FUNCTION_BLOCK TcoSequencerAutoRestorableTest EXTENDS TcoCore._internals_TcoContext
VAR
	_callMyPlcInstance	:	BOOL := FALSE;
	_sequencer : _TcoSequencer(THIS^, NO.Structure, eRestoreMode.AutoRestoreMembers);
	_runPLCinstanceOnce : BOOL := FALSE;
	_runPLCinstanceCyclicaly : BOOL := FALSE;
	_stepID : INT := 32764;
	_enabled : BOOL;
	_stepDescription : STRING := 'Last step sequence message';	
	_runOneStep : BOOL;
	_runAllSteps : BOOL;
	_finishStep : BOOL;
	_restore : BOOL;
	_cycleCount : INT;
	_restoreCycleCount : INT;
	_init: BOOL;
	_setCurrentStepPropTestData : TcoCore.StepDetails;
END_VAR

IF _callMyPlcInstance THEN
	IF NOT _init THEN
		ContextOpen();	
		ContextClose();	
		_init := THIS^._rtc.IsValid;
	END_IF
	
	IF _restore THEN
		ContextOpen();	
		THIS^._sequencer.Restore();	
		_restoreCycleCount := _restoreCycleCount + 1;
		_restore := FALSE;
		ContextClose();	
		RETURN;
	END_IF
	
	IF _runPLCinstanceOnce AND NOT _runPLCinstanceCyclicaly THEN
		ContextOpen();	
		THIS^.PLCinstanceRun(_stepID , _enabled, _stepDescription);
		_cycleCount := _cycleCount + 1;
		_runPLCinstanceOnce := FALSE;
		ContextClose();	
	END_IF
	
	IF _runPLCinstanceCyclicaly AND NOT _runPLCinstanceOnce THEN
		ContextOpen();	
		THIS^.PLCinstanceRun(_stepID , _enabled, _stepDescription);
		_cycleCount := _cycleCount + 1;
		ContextClose();	
	END_IF
END_IF;

{attribute 'TcRpcEnable'}
METHOD ChildHasAutoRestoreEnabled : BOOL;
ChildHasAutoRestoreEnabled := _sequencer.ChildHasAutoRestoreEnabled();
END_METHOD

{attribute 'TcRpcEnable'}
METHOD ChildIsAutoRestorable : BOOL;
ChildIsAutoRestorable := _sequencer.ChildIsAutoRestorable();
END_METHOD

{attribute 'TcRpcEnable'}
METHOD CleanupPointers
_sequencer.CleanupPointers();
END_METHOD

{attribute 'TcRpcEnable'}
METHOD ClearNumberOfSteps
_sequencer.ClearNumberOfSteps();
END_METHOD

{attribute 'TcRpcEnable'}
METHOD PROTECTED ContextClose
SUPER^._Close();
END_METHOD

{attribute 'TcRpcEnable'}
METHOD ContextOpen
SUPER^._Open();
END_METHOD

{attribute 'TcRpcEnable'}
METHOD GetChildState : INT
GetChildState := _sequencer.GetChildState();
END_METHOD

{attribute 'TcRpcEnable'}
METHOD GetCurrentStepOrder : UINT
GetCurrentStepOrder := _sequencer._currentStep.Order;
END_METHOD

{attribute 'TcRpcEnable'}
METHOD GetCurrentStepPropTest
_setCurrentStepPropTestData := THIS^._sequencer.CurrentStep;
END_METHOD

{attribute 'TcRpcEnable'}
METHOD GetNumberOfStepsInSequence : UINT
GetNumberOfStepsInSequence := _sequencer._numberOfStepsInSequence;
END_METHOD

{attribute 'TcRpcEnable'}
METHOD GetOrderOfTheCurrentlyEvaluatedStep : UINT
GetOrderOfTheCurrentlyEvaluatedStep := _sequencer._theOrderOfTheCurrentlyEvaluatedStep;
END_METHOD

{attribute 'TcRpcEnable'}
METHOD GetOrderOfTheCurrentlyExecutedStep : UINT
GetOrderOfTheCurrentlyExecutedStep := _sequencer._theOrderOfTheCurrentlyExecutedStep;
END_METHOD

{attribute 'TcRpcEnable'}
METHOD GetPreviousNumberOfStepsInSequence : UINT
GetPreviousNumberOfStepsInSequence := _sequencer._previousNumberOfStepsInSequence;
END_METHOD

{attribute 'TcRpcEnable'}
METHOD GetRequestStepCycle : UINT
GetRequestStepCycle := _sequencer.RequestStepCycle;
END_METHOD

{attribute 'TcRpcEnable'}
METHOD GetSequencerErrorId : INT
GetSequencerErrorId := _sequencer.GetSequencerErrorId();
END_METHOD

{attribute 'TcRpcEnable'}
METHOD GetTextOfTheMostImportantMessage : STRING(254)
GetTextOfTheMostImportantMessage := THIS^._sequencer.GetTextOfTheMostImportantMessage();
END_METHOD

{attribute 'TcRpcEnable'}
METHOD HasAutoRestoreEnabled : BOOL;
HasAutoRestoreEnabled := _sequencer.HasAutoRestoreEnabled();
END_METHOD

{attribute 'TcRpcEnable'}
METHOD IsAutoRestorable : BOOL;
IsAutoRestorable := _sequencer.IsAutoRestorable();
END_METHOD

{attribute 'TcRpcEnable'}
METHOD IsFirstStepEntry : BOOL
IsFirstStepEntry := THIS^._sequencer.IsFirstStepEntry();
END_METHOD

METHOD PROTECTED  Main
END_METHOD

{attribute 'TcRpcEnable'}
METHOD PLCinstanceRun
VAR_INPUT
	inStepId			:	UINT;
	inEnabled			:	BOOL;
	inStepDescription	:	STRING(254);	
END_VAR
THIS^._sequencer.SetTestParams(	_runOneStep , _runAllSteps , _finishStep , inStepId , inEnabled , inStepDescription);

THIS^._sequencer.Run();
END_METHOD

{attribute 'TcRpcEnable'}
METHOD RequestStep
VAR_INPUT
	inRequestedStepId : INT;
END_VAR
_sequencer._RequestStep(inRequestedStepId);
END_METHOD

{attribute 'TcRpcEnable'}
METHOD Restore
_sequencer.Restore();
END_METHOD

{attribute 'TcRpcEnable'}
METHOD SequenceComplete
_sequencer._SequenceComplete();
END_METHOD

{attribute 'TcRpcEnable'}
METHOD SequencerClose
THIS^._sequencer.SequencerClose();
END_METHOD

{attribute 'TcRpcEnable'}
METHOD SequencerHasError : BOOL
SequencerHasError := _sequencer.SequencerHasError();
END_METHOD

{attribute 'TcRpcEnable'}
METHOD SequencerOpen
THIS^._sequencer.SequencerOpen();
END_METHOD

{attribute 'TcRpcEnable'}
METHOD SetChildState
VAR_INPUT
	inState			:	INT;
END_VAR
_sequencer.SetChildState(inState);
END_METHOD

{attribute 'TcRpcEnable'}
METHOD SetCurrentStep
VAR_INPUT
	inStepID 			:	INT;
	inStepDescription	:	STRING(254);
END_VAR
_sequencer.SetCurrentStep(inStepID := inStepID, inStepDescription := inStepDescription);
END_METHOD

{attribute 'TcRpcEnable'}
METHOD SetCurrentStepToErrorState : BOOL
SetCurrentStepToErrorState := _sequencer.SetCurrentStepToErrorState();
END_METHOD

{attribute 'TcRpcEnable'}
METHOD SetCyclicMode : BOOL
SetCyclicMode := _sequencer.SetCyclicMode();
END_METHOD

{attribute 'TcRpcEnable'}
METHOD SetInvalidMode : BOOL
SetInvalidMode := _sequencer.SetInvalidMode();
END_METHOD

{attribute 'TcRpcEnable'}
METHOD SetNumberOfSteps : UINT
VAR_INPUT
	inNumberOfSteps :UINT;
END_VAR
_sequencer.SetNumberOfSteps(inNumberOfSteps);
SetNumberOfSteps := _sequencer._numberOfStepsInSequence;
END_METHOD

{attribute 'TcRpcEnable'}
METHOD SetRequestStepCycle : UINT
VAR_INPUT
	Value : UINT;
END_VAR
_sequencer.RequestStepCycle := Value;

SetRequestStepCycle := _sequencer.RequestStepCycle;
END_METHOD

{attribute 'TcRpcEnable'}
METHOD SetSequenceAsChecked : BOOL
VAR_INPUT
END_VAR
_sequencer.SetSequenceAsChecked();
END_METHOD

{attribute 'TcRpcEnable'}
METHOD SetSequenceAsNotChecked : BOOL
VAR_INPUT
END_VAR
_sequencer.SetSequenceAsNotChecked();
END_METHOD

{attribute 'TcRpcEnable'}
METHOD SetStepMode : BOOL
SetStepMode := _sequencer.SetStepMode();
END_METHOD

{attribute 'TcRpcEnable'}
METHOD Step : BOOL
VAR_INPUT
	inStepId			:	INT;
	inEnabled			:	BOOL;
	inStepDescription	:	STRING(254);		
END_VAR
Step := _sequencer._Step(inStepID := inStepId, inEnabled := inEnabled, inStepDescription := inStepDescription);
END_METHOD

{attribute 'TcRpcEnable'}
METHOD StepBackward
_sequencer._StepBackward();
END_METHOD

{attribute 'TcRpcEnable'}
METHOD StepCompleteWhen 
VAR_INPUT
	inCondition : BOOL;
END_VAR
_sequencer._StepCompleteWhen(inCondition);
END_METHOD

{attribute 'TcRpcEnable'}
METHOD StepForward
_sequencer._StepForward();
END_METHOD

{attribute 'TcRpcEnable'}
METHOD StepIn
_sequencer._StepIn();
END_METHOD

{attribute 'TcRpcEnable'}
METHOD UpdateCurrentStepDetails
VAR_INPUT
END_VAR
_sequencer.UpdateCurrentStepDetails();
END_METHOD

END_FUNCTION_BLOCK

(* stored: Version 1.1.0.1
   POU TcoSequencerAutoRestorableTest: Id {562bb59c-4938-0c9c-3dbf-3bf62db74778}, SpecialFunc None
   Method ChildHasAutoRestoreEnabled: Id {c5f7e550-1c06-02b1-3dc1-0350c51bf48f}
   Method ChildIsAutoRestorable: Id {5f9d102f-a62b-0055-03e2-11e38b840327}
   Method CleanupPointers: Id {14bc8b6e-cfa4-0753-0342-ac2726e5612b}
   Method ClearNumberOfSteps: Id {f539a6b0-7bc6-0301-3239-7213868811cf}
   Method ContextClose: Id {810ef247-629a-0b8d-2e62-074f616b849f}
   Method ContextOpen: Id {74cc42e7-8072-0180-190b-77d20dffc054}
   Method GetChildState: Id {1698e5e7-e8f6-0d10-2e8a-504f2dba89f9}
   Method GetCurrentStepOrder: Id {705846ff-2eb1-0e94-0c3d-3991277063da}
   Method GetCurrentStepPropTest: Id {66619082-c818-04f9-2a66-526f96036c15}
   Method GetNumberOfStepsInSequence: Id {9788b597-1936-060b-27fc-789b2bcb0619}
   Method GetOrderOfTheCurrentlyEvaluatedStep: Id {7364c59e-c7f0-090d-2cf6-5ee61adf64f1}
   Method GetOrderOfTheCurrentlyExecutedStep: Id {7a373085-9eff-0d2d-02ce-b9d12b15a209}
   Method GetPreviousNumberOfStepsInSequence: Id {e3e2f302-0f06-088b-105b-80cc8ce26fe8}
   Method GetRequestStepCycle: Id {6131ad9e-58e1-0a8f-2ab1-5fc68e9d6d51}
   Method GetSequencerErrorId: Id {b86191c5-a461-08a6-156b-3245d5b8cd08}
   Method GetTextOfTheMostImportantMessage: Id {2ed534f1-5f3c-0f0a-0d20-164428a174da}
   Method HasAutoRestoreEnabled: Id {36504de3-bf07-0b24-007a-e5676ed071a7}
   Method IsAutoRestorable: Id {cfba587a-0b0d-065c-2f47-ce74088893ee}
   Method IsFirstStepEntry: Id {c14a3461-1c50-0d1d-04c7-d0042dce9c24}
   Method Main: Id {4b8637ef-642e-0b3e-3e8b-c3b3127d9586}
   Method PLCinstanceRun: Id {efc71d82-94d5-06e4-2e8c-904a97b90c09}
   Method RequestStep: Id {d064fc61-7128-02aa-26bf-bd5b5c4a4123}
   Method Restore: Id {74637749-b130-086a-1666-3cbc30d0057d}
   Method SequenceComplete: Id {a191839d-c590-0f09-2cf6-c8c146585bce}
   Method SequencerClose: Id {6b1546d7-64aa-0b4d-1d11-f840a931f4d2}
   Method SequencerHasError: Id {e9d487eb-3da5-0ed0-342c-3acceaff3d30}
   Method SequencerOpen: Id {6c2f6e39-03f9-0b02-17d0-cea8266bae99}
   Method SetChildState: Id {d5a0f8e4-3788-06d6-27cb-c53d0981f0ec}
   Method SetCurrentStep: Id {55cbe96f-cdad-0ac3-2572-19e947b68eea}
   Method SetCurrentStepToErrorState: Id {ad88f54b-d3fd-0a42-09c6-aae6e1520a2e}
   Method SetCyclicMode: Id {e977a0e7-185a-07bd-29a5-b65af2291fa7}
   Method SetInvalidMode: Id {c68ce154-b258-0796-3a54-6339ebb459ae}
   Method SetNumberOfSteps: Id {deae86d4-9245-0599-14b1-6cd3be2fc100}
   Method SetRequestStepCycle: Id {320a475c-59fb-060c-1340-c1cd47565189}
   Method SetSequenceAsChecked: Id {8f4ed25a-c856-0939-3141-83567ffa79af}
   Method SetSequenceAsNotChecked: Id {a4a33e8e-a4c2-0e71-3d3c-3b5837d7e9e0}
   Method SetStepMode: Id {0cbf1bb4-7bfb-03c0-121b-e84f9c762f04}
   Method Step: Id {36dc7d2f-60ca-09f7-1ca1-b698678bf81b}
   Method StepBackward: Id {efaa54c3-3ad2-0cc0-1bfc-95f39d7fc5fc}
   Method StepCompleteWhen: Id {748eaa1c-8971-0692-12bd-ab735fc9acd3}
   Method StepForward: Id {7d0da0d7-526d-0f81-2a51-0285e61cfeec}
   Method StepIn: Id {ef1cc9f2-d06b-08b3-0511-a8c62d15235c}
   Method UpdateCurrentStepDetails: Id {dee5e4a8-6675-06d9-2524-11319c1dcd1a} *)
